// TIA Portal V17 export
// export: Created 2024-08-07T21:44:00.3831212Z, ExportSetting WithDefaults, DisplayName Totally Integrated Automation Portal, DisplayVersion V17 Update 7, DisplayName TIA Portal Openness, DisplayVersion V17 Update 7, DisplayName TIA Portal Version Control Interface, DisplayVersion V17, DisplayName SINAMICS Startdrive Advanced, DisplayVersion V17 SP2, DisplayName SINAMICS Startdrive G110M, G120, G120C, G120D, G120P, G115D, DisplayVersion V17 SP2, DisplayName SINAMICS Startdrive G130, G150, S120, S150, SINAMICS MV, S210, DisplayVersion V17 SP2, DisplayName STEP 7 Professional, DisplayVersion V17 Update 7, DisplayName STEP 7 Safety, DisplayVersion V17 Update 6, DisplayName WinCC Advanced / Unified PC, DisplayVersion V17 Update 7
DATA_BLOCK "DB_EksList"   // DB5051
{ S7_Optimized_Access := 'TRUE' }
VERSION : 0.1
// stored: AutoNumber false, DBAccessibleFromOPCUA true, DBAccessibleFromWebserver true, IsOnlyStoredInLoadMemory false, IsRetainMemResEnabled false, IsWriteProtectedInAS false, MemoryReserve 100
   VAR RETAIN
      Key { S7_SetPoint := 'True'} : Array[1.."EksNumberOfKeys"] of "UDT_EksKey";
   END_VAR
BEGIN
   Key[1..5].Level := 5;
   Key[6..9].Level := 3;
   Key[10..13].Level := 2;
   Key[14..18].Level := 5;
   Key[19..100].Level := 0;
   Key[1].EmployeeID[1..4] := ' ';
   Key[2].EmployeeID[1] := '¥';
   Key[2].EmployeeID[2] := 'Z';
   Key[2].EmployeeID[3] := '¥';
   Key[2].EmployeeID[4] := 'Z';
   Key[3].EmployeeID[1..4] := ' ';
   Key[4].EmployeeID[1..4] := ' ';
   Key[5].EmployeeID[1..4] := ' ';
   Key[6].EmployeeID[1..4] := ' ';
   Key[7].EmployeeID[1..4] := ' ';
   Key[8].EmployeeID[1..4] := ' ';
   Key[9].EmployeeID[1..4] := ' ';
   Key[10].EmployeeID[1..4] := ' ';
   Key[11].EmployeeID[1..4] := ' ';
   Key[12].EmployeeID[1..4] := ' ';
   Key[13].EmployeeID[1..4] := ' ';
   Key[14].EmployeeID[1..4] := ' ';
   Key[15].EmployeeID[1..4] := ' ';
   Key[16].EmployeeID[1..4] := ' ';
   Key[17].EmployeeID[1..4] := ' ';
   Key[18].EmployeeID[1..4] := ' ';
   Key[19].EmployeeID[1..4] := ' ';
   Key[20].EmployeeID[1..4] := ' ';
   Key[21].EmployeeID[1..4] := ' ';
   Key[22].EmployeeID[1..4] := ' ';
   Key[23].EmployeeID[1..4] := ' ';
   Key[24].EmployeeID[1..4] := ' ';
   Key[25].EmployeeID[1..4] := ' ';
   Key[26].EmployeeID[1..4] := ' ';
   Key[27].EmployeeID[1..4] := ' ';
   Key[28].EmployeeID[1..4] := ' ';
   Key[29].EmployeeID[1..4] := ' ';
   Key[30].EmployeeID[1..4] := ' ';
   Key[31].EmployeeID[1..4] := ' ';
   Key[32].EmployeeID[1..4] := ' ';
   Key[33].EmployeeID[1..4] := ' ';
   Key[34].EmployeeID[1..4] := ' ';
   Key[35].EmployeeID[1..4] := ' ';
   Key[36].EmployeeID[1..4] := ' ';
   Key[37].EmployeeID[1..4] := ' ';
   Key[38].EmployeeID[1..4] := ' ';
   Key[39].EmployeeID[1..4] := ' ';
   Key[40].EmployeeID[1..4] := ' ';
   Key[41].EmployeeID[1..4] := ' ';
   Key[42].EmployeeID[1..4] := ' ';
   Key[43].EmployeeID[1..4] := ' ';
   Key[44].EmployeeID[1..4] := ' ';
   Key[45].EmployeeID[1..4] := ' ';
   Key[46].EmployeeID[1..4] := ' ';
   Key[47].EmployeeID[1..4] := ' ';
   Key[48].EmployeeID[1..4] := ' ';
   Key[49].EmployeeID[1..4] := ' ';
   Key[50].EmployeeID[1..4] := ' ';
   Key[51].EmployeeID[1..4] := ' ';
   Key[52].EmployeeID[1..4] := ' ';
   Key[53].EmployeeID[1..4] := ' ';
   Key[54].EmployeeID[1..4] := ' ';
   Key[55].EmployeeID[1..4] := ' ';
   Key[56].EmployeeID[1..4] := ' ';
   Key[57].EmployeeID[1..4] := ' ';
   Key[58].EmployeeID[1..4] := ' ';
   Key[59].EmployeeID[1..4] := ' ';
   Key[60].EmployeeID[1..4] := ' ';
   Key[61].EmployeeID[1..4] := ' ';
   Key[62].EmployeeID[1..4] := ' ';
   Key[63].EmployeeID[1..4] := ' ';
   Key[64].EmployeeID[1..4] := ' ';
   Key[65].EmployeeID[1..4] := ' ';
   Key[66].EmployeeID[1..4] := ' ';
   Key[67].EmployeeID[1..4] := ' ';
   Key[68].EmployeeID[1..4] := ' ';
   Key[69].EmployeeID[1..4] := ' ';
   Key[70].EmployeeID[1..4] := ' ';
   Key[71].EmployeeID[1..4] := ' ';
   Key[72].EmployeeID[1..4] := ' ';
   Key[73].EmployeeID[1..4] := ' ';
   Key[74].EmployeeID[1..4] := ' ';
   Key[75].EmployeeID[1..4] := ' ';
   Key[76].EmployeeID[1..4] := ' ';
   Key[77].EmployeeID[1..4] := ' ';
   Key[78].EmployeeID[1..4] := ' ';
   Key[79].EmployeeID[1..4] := ' ';
   Key[80].EmployeeID[1..4] := ' ';
   Key[81].EmployeeID[1..4] := ' ';
   Key[82].EmployeeID[1..4] := ' ';
   Key[83].EmployeeID[1..4] := ' ';
   Key[84].EmployeeID[1..4] := ' ';
   Key[85].EmployeeID[1..4] := ' ';
   Key[86].EmployeeID[1..4] := ' ';
   Key[87].EmployeeID[1..4] := ' ';
   Key[88].EmployeeID[1..4] := ' ';
   Key[89].EmployeeID[1..4] := ' ';
   Key[90].EmployeeID[1..4] := ' ';
   Key[91].EmployeeID[1..4] := ' ';
   Key[92].EmployeeID[1..4] := ' ';
   Key[93].EmployeeID[1..4] := ' ';
   Key[94].EmployeeID[1..4] := ' ';
   Key[95].EmployeeID[1..4] := ' ';
   Key[96].EmployeeID[1..4] := ' ';
   Key[97].EmployeeID[1..4] := ' ';
   Key[98].EmployeeID[1..4] := ' ';
   Key[99].EmployeeID[1..4] := ' ';
   Key[100].EmployeeID[1..4] := ' ';
   Key[1].KeyID[1] := '0';
   Key[1].KeyID[2] := '3';
   Key[1].KeyID[3] := '6';
   Key[1].KeyID[4] := 'C';
   Key[1].KeyID[5] := 'B';
   Key[1].KeyID[6] := 'C';
   Key[1].KeyID[7] := 'F';
   Key[1].KeyID[8] := '4';
   Key[1].KeyID[9] := '0';
   Key[1].KeyID[10] := 'F';
   Key[1].KeyID[11..12] := '0';
   Key[1].KeyID[13] := '1';
   Key[1].KeyID[14] := '0';
   Key[1].KeyID[15] := '3';
   Key[1].KeyID[16] := '2';
   Key[2].KeyID[1] := '0';
   Key[2].KeyID[2..3] := '3';
   Key[2].KeyID[4] := 'E';
   Key[2].KeyID[5] := '0';
   Key[2].KeyID[6] := '2';
   Key[2].KeyID[7] := 'E';
   Key[2].KeyID[8] := '5';
   Key[2].KeyID[9] := 'C';
   Key[2].KeyID[10] := 'B';
   Key[2].KeyID[11..12] := '0';
   Key[2].KeyID[13] := '1';
   Key[2].KeyID[14] := '0';
   Key[2].KeyID[15] := '3';
   Key[2].KeyID[16] := '2';
   Key[3].KeyID[1] := '0';
   Key[3].KeyID[2] := '3';
   Key[3].KeyID[3] := '7';
   Key[3].KeyID[4] := '2';
   Key[3].KeyID[5] := '4';
   Key[3].KeyID[6] := '5';
   Key[3].KeyID[7] := '2';
   Key[3].KeyID[8] := '9';
   Key[3].KeyID[9] := 'A';
   Key[3].KeyID[10] := '6';
   Key[3].KeyID[11..12] := '0';
   Key[3].KeyID[13] := '1';
   Key[3].KeyID[14] := '0';
   Key[3].KeyID[15] := '3';
   Key[3].KeyID[16] := '2';
   Key[4].KeyID[1] := '0';
   Key[4].KeyID[2] := '3';
   Key[4].KeyID[3] := '7';
   Key[4].KeyID[4] := '2';
   Key[4].KeyID[5..6] := '5';
   Key[4].KeyID[7] := '9';
   Key[4].KeyID[8] := 'D';
   Key[4].KeyID[9] := '8';
   Key[4].KeyID[10] := 'A';
   Key[4].KeyID[11..12] := '0';
   Key[4].KeyID[13] := '1';
   Key[4].KeyID[14] := '0';
   Key[4].KeyID[15] := '3';
   Key[4].KeyID[16] := '2';
   Key[5].KeyID[1] := '0';
   Key[5].KeyID[2] := '3';
   Key[5].KeyID[3] := '7';
   Key[5].KeyID[4] := '2';
   Key[5].KeyID[5] := '4';
   Key[5].KeyID[6] := '3';
   Key[5].KeyID[7] := 'B';
   Key[5].KeyID[8] := 'A';
   Key[5].KeyID[9] := '3';
   Key[5].KeyID[10] := 'F';
   Key[5].KeyID[11..12] := '0';
   Key[5].KeyID[13] := '1';
   Key[5].KeyID[14] := '0';
   Key[5].KeyID[15] := '3';
   Key[5].KeyID[16] := '2';
   Key[6].KeyID[1] := '0';
   Key[6].KeyID[2] := '3';
   Key[6].KeyID[3] := '7';
   Key[6].KeyID[4] := '2';
   Key[6].KeyID[5] := '9';
   Key[6].KeyID[6] := '7';
   Key[6].KeyID[7] := '0';
   Key[6].KeyID[8] := 'C';
   Key[6].KeyID[9] := '2';
   Key[6].KeyID[10] := 'A';
   Key[6].KeyID[11..12] := '0';
   Key[6].KeyID[13] := '1';
   Key[6].KeyID[14] := '0';
   Key[6].KeyID[15] := '3';
   Key[6].KeyID[16] := '2';
   Key[7].KeyID[1] := '0';
   Key[7].KeyID[2] := '3';
   Key[7].KeyID[3] := '7';
   Key[7].KeyID[4] := '3';
   Key[7].KeyID[5] := '0';
   Key[7].KeyID[6] := 'A';
   Key[7].KeyID[7] := 'D';
   Key[7].KeyID[8] := '7';
   Key[7].KeyID[9] := '0';
   Key[7].KeyID[10] := '1';
   Key[7].KeyID[11..12] := '0';
   Key[7].KeyID[13] := '1';
   Key[7].KeyID[14] := '0';
   Key[7].KeyID[15] := '3';
   Key[7].KeyID[16] := '2';
   Key[8].KeyID[1] := '0';
   Key[8].KeyID[2] := '3';
   Key[8].KeyID[3] := '7';
   Key[8].KeyID[4] := '2';
   Key[8].KeyID[5] := '4';
   Key[8].KeyID[6..7] := '5';
   Key[8].KeyID[8..9] := 'F';
   Key[8].KeyID[10] := 'B';
   Key[8].KeyID[11..12] := '0';
   Key[8].KeyID[13] := '1';
   Key[8].KeyID[14] := '0';
   Key[8].KeyID[15] := '3';
   Key[8].KeyID[16] := '2';
   Key[9].KeyID[1] := '0';
   Key[9].KeyID[2] := '3';
   Key[9].KeyID[3] := '7';
   Key[9].KeyID[4] := '2';
   Key[9].KeyID[5] := '9';
   Key[9].KeyID[6] := 'C';
   Key[9].KeyID[7] := '3';
   Key[9].KeyID[8] := '8';
   Key[9].KeyID[9] := '3';
   Key[9].KeyID[10] := '2';
   Key[9].KeyID[11..12] := '0';
   Key[9].KeyID[13] := '1';
   Key[9].KeyID[14] := '0';
   Key[9].KeyID[15] := '3';
   Key[9].KeyID[16] := '2';
   Key[10].KeyID[1] := '0';
   Key[10].KeyID[2] := '3';
   Key[10].KeyID[3] := '7';
   Key[10].KeyID[4] := '2';
   Key[10].KeyID[5] := 'C';
   Key[10].KeyID[6..7] := '3';
   Key[10].KeyID[8] := 'E';
   Key[10].KeyID[9] := 'B';
   Key[10].KeyID[10] := '6';
   Key[10].KeyID[11..12] := '0';
   Key[10].KeyID[13] := '1';
   Key[10].KeyID[14] := '0';
   Key[10].KeyID[15] := '3';
   Key[10].KeyID[16] := '2';
   Key[11].KeyID[1] := '0';
   Key[11].KeyID[2] := '3';
   Key[11].KeyID[3] := '7';
   Key[11].KeyID[4] := '3';
   Key[11].KeyID[5] := '0';
   Key[11].KeyID[6] := 'C';
   Key[11].KeyID[7] := '3';
   Key[11].KeyID[8] := '0';
   Key[11].KeyID[9] := 'B';
   Key[11].KeyID[10] := 'F';
   Key[11].KeyID[11..12] := '0';
   Key[11].KeyID[13] := '1';
   Key[11].KeyID[14] := '0';
   Key[11].KeyID[15] := '3';
   Key[11].KeyID[16] := '2';
   Key[12].KeyID[1] := '0';
   Key[12].KeyID[2] := '3';
   Key[12].KeyID[3] := '7';
   Key[12].KeyID[4] := '2';
   Key[12].KeyID[5] := 'F';
   Key[12].KeyID[6] := '4';
   Key[12].KeyID[7] := 'D';
   Key[12].KeyID[8] := 'F';
   Key[12].KeyID[9] := '5';
   Key[12].KeyID[10] := 'C';
   Key[12].KeyID[11..12] := '0';
   Key[12].KeyID[13] := '1';
   Key[12].KeyID[14] := '0';
   Key[12].KeyID[15] := '3';
   Key[12].KeyID[16] := '2';
   Key[13].KeyID[1] := '0';
   Key[13].KeyID[2] := '3';
   Key[13].KeyID[3] := '7';
   Key[13].KeyID[4] := '2';
   Key[13].KeyID[5] := 'C';
   Key[13].KeyID[6] := '9';
   Key[13].KeyID[7] := '1';
   Key[13].KeyID[8..9] := '6';
   Key[13].KeyID[10] := '7';
   Key[13].KeyID[11..12] := '0';
   Key[13].KeyID[13] := '1';
   Key[13].KeyID[14] := '0';
   Key[13].KeyID[15] := '3';
   Key[13].KeyID[16] := '2';
   Key[14].KeyID[1] := '0';
   Key[14].KeyID[2] := '3';
   Key[14].KeyID[3] := '2';
   Key[14].KeyID[4] := '3';
   Key[14].KeyID[5] := 'C';
   Key[14].KeyID[6] := 'F';
   Key[14].KeyID[7] := '5';
   Key[14].KeyID[8] := 'E';
   Key[14].KeyID[9..10] := 'B';
   Key[14].KeyID[11..12] := '0';
   Key[14].KeyID[13] := '1';
   Key[14].KeyID[14] := '0';
   Key[14].KeyID[15] := '3';
   Key[14].KeyID[16] := '2';
   Key[15].KeyID[1] := '0';
   Key[15].KeyID[2] := '3';
   Key[15].KeyID[3] := '6';
   Key[15].KeyID[4] := '1';
   Key[15].KeyID[5] := 'E';
   Key[15].KeyID[6] := '8';
   Key[15].KeyID[7] := '1';
   Key[15].KeyID[8] := '4';
   Key[15].KeyID[9] := 'A';
   Key[15].KeyID[10] := 'E';
   Key[15].KeyID[11..12] := '0';
   Key[15].KeyID[13] := '1';
   Key[15].KeyID[14] := '0';
   Key[15].KeyID[15] := '3';
   Key[15].KeyID[16] := '2';
   Key[16].KeyID[1] := '0';
   Key[16].KeyID[2] := '3';
   Key[16].KeyID[3] := '7';
   Key[16].KeyID[4] := '1';
   Key[16].KeyID[5] := 'E';
   Key[16].KeyID[6] := 'D';
   Key[16].KeyID[7] := '1';
   Key[16].KeyID[8] := '2';
   Key[16].KeyID[9] := 'B';
   Key[16].KeyID[10] := '7';
   Key[16].KeyID[11..12] := '0';
   Key[16].KeyID[13] := '1';
   Key[16].KeyID[14] := '0';
   Key[16].KeyID[15] := '3';
   Key[16].KeyID[16] := '2';
   Key[17].KeyID[1] := '0';
   Key[17].KeyID[2] := '3';
   Key[17].KeyID[3] := '7';
   Key[17].KeyID[4] := '2';
   Key[17].KeyID[5] := 'F';
   Key[17].KeyID[6] := '5';
   Key[17].KeyID[7] := '2';
   Key[17].KeyID[8] := 'C';
   Key[17].KeyID[9] := '6';
   Key[17].KeyID[10] := '8';
   Key[17].KeyID[11..12] := '0';
   Key[17].KeyID[13] := '1';
   Key[17].KeyID[14] := '0';
   Key[17].KeyID[15] := '3';
   Key[17].KeyID[16] := '2';
   Key[18].KeyID[1] := '0';
   Key[18].KeyID[2] := '3';
   Key[18].KeyID[3] := '7';
   Key[18].KeyID[4] := '1';
   Key[18].KeyID[5..7] := 'F';
   Key[18].KeyID[8] := 'C';
   Key[18].KeyID[9] := '4';
   Key[18].KeyID[10] := '2';
   Key[18].KeyID[11..12] := '0';
   Key[18].KeyID[13] := '1';
   Key[18].KeyID[14] := '0';
   Key[18].KeyID[15] := '3';
   Key[18].KeyID[16] := '2';
   Key[19].KeyID[1..16] := ' ';
   Key[20].KeyID[1..16] := ' ';
   Key[21].KeyID[1..16] := ' ';
   Key[22].KeyID[1..16] := ' ';
   Key[23].KeyID[1..16] := ' ';
   Key[24].KeyID[1..16] := ' ';
   Key[25].KeyID[1..16] := ' ';
   Key[26].KeyID[1..16] := ' ';
   Key[27].KeyID[1..16] := ' ';
   Key[28].KeyID[1..16] := ' ';
   Key[29].KeyID[1..16] := ' ';
   Key[30].KeyID[1..16] := ' ';
   Key[31].KeyID[1..16] := ' ';
   Key[32].KeyID[1..16] := ' ';
   Key[33].KeyID[1..16] := ' ';
   Key[34].KeyID[1..16] := ' ';
   Key[35].KeyID[1..16] := ' ';
   Key[36].KeyID[1..16] := ' ';
   Key[37].KeyID[1..16] := ' ';
   Key[38].KeyID[1..16] := ' ';
   Key[39].KeyID[1..16] := ' ';
   Key[40].KeyID[1..16] := ' ';
   Key[41].KeyID[1..16] := ' ';
   Key[42].KeyID[1..16] := ' ';
   Key[43].KeyID[1..16] := ' ';
   Key[44].KeyID[1..16] := ' ';
   Key[45].KeyID[1..16] := ' ';
   Key[46].KeyID[1..16] := ' ';
   Key[47].KeyID[1..16] := ' ';
   Key[48].KeyID[1..16] := ' ';
   Key[49].KeyID[1..16] := ' ';
   Key[50].KeyID[1..16] := ' ';
   Key[51].KeyID[1..16] := ' ';
   Key[52].KeyID[1..16] := ' ';
   Key[53].KeyID[1..16] := ' ';
   Key[54].KeyID[1..16] := ' ';
   Key[55].KeyID[1..16] := ' ';
   Key[56].KeyID[1..16] := ' ';
   Key[57].KeyID[1..16] := ' ';
   Key[58].KeyID[1..16] := ' ';
   Key[59].KeyID[1..16] := ' ';
   Key[60].KeyID[1..16] := ' ';
   Key[61].KeyID[1..16] := ' ';
   Key[62].KeyID[1..16] := ' ';
   Key[63].KeyID[1..16] := ' ';
   Key[64].KeyID[1..16] := ' ';
   Key[65].KeyID[1..16] := ' ';
   Key[66].KeyID[1..16] := ' ';
   Key[67].KeyID[1..16] := ' ';
   Key[68].KeyID[1..16] := ' ';
   Key[69].KeyID[1..16] := ' ';
   Key[70].KeyID[1..16] := ' ';
   Key[71].KeyID[1..16] := ' ';
   Key[72].KeyID[1..16] := ' ';
   Key[73].KeyID[1..16] := ' ';
   Key[74].KeyID[1..16] := ' ';
   Key[75].KeyID[1..16] := ' ';
   Key[76].KeyID[1..16] := ' ';
   Key[77].KeyID[1..16] := ' ';
   Key[78].KeyID[1..16] := ' ';
   Key[79].KeyID[1..16] := ' ';
   Key[80].KeyID[1..16] := ' ';
   Key[81].KeyID[1..16] := ' ';
   Key[82].KeyID[1..16] := ' ';
   Key[83].KeyID[1..16] := ' ';
   Key[84].KeyID[1..16] := ' ';
   Key[85].KeyID[1..16] := ' ';
   Key[86].KeyID[1..16] := ' ';
   Key[87].KeyID[1..16] := ' ';
   Key[88].KeyID[1..16] := ' ';
   Key[89].KeyID[1..16] := ' ';
   Key[90].KeyID[1..16] := ' ';
   Key[91].KeyID[1..16] := ' ';
   Key[92].KeyID[1..16] := ' ';
   Key[93].KeyID[1..16] := ' ';
   Key[94].KeyID[1..16] := ' ';
   Key[95].KeyID[1..16] := ' ';
   Key[96].KeyID[1..16] := ' ';
   Key[97].KeyID[1..16] := ' ';
   Key[98].KeyID[1..16] := ' ';
   Key[99].KeyID[1..16] := ' ';
   Key[100].KeyID[1..16] := ' ';
   Key[1].Comment[1..20] := ' ';
   Key[2].Comment[1..20] := ' ';
   Key[3].Comment[1..20] := ' ';
   Key[4].Comment[1..20] := ' ';
   Key[5].Comment[1..20] := ' ';
   Key[6].Comment[1..20] := ' ';
   Key[7].Comment[1..20] := ' ';
   Key[8].Comment[1..20] := ' ';
   Key[9].Comment[1..20] := ' ';
   Key[10].Comment[1..20] := ' ';
   Key[11].Comment[1..20] := ' ';
   Key[12].Comment[1..20] := ' ';
   Key[13].Comment[1..20] := ' ';
   Key[14].Comment[1..20] := ' ';
   Key[15].Comment[1..20] := ' ';
   Key[16].Comment[1..20] := ' ';
   Key[17].Comment[1..20] := ' ';
   Key[18].Comment[1..20] := ' ';
   Key[19].Comment[1..20] := ' ';
   Key[20].Comment[1..20] := ' ';
   Key[21].Comment[1..20] := ' ';
   Key[22].Comment[1..20] := ' ';
   Key[23].Comment[1..20] := ' ';
   Key[24].Comment[1..20] := ' ';
   Key[25].Comment[1..20] := ' ';
   Key[26].Comment[1..20] := ' ';
   Key[27].Comment[1..20] := ' ';
   Key[28].Comment[1..20] := ' ';
   Key[29].Comment[1..20] := ' ';
   Key[30].Comment[1..20] := ' ';
   Key[31].Comment[1..20] := ' ';
   Key[32].Comment[1..20] := ' ';
   Key[33].Comment[1..20] := ' ';
   Key[34].Comment[1..20] := ' ';
   Key[35].Comment[1..20] := ' ';
   Key[36].Comment[1..20] := ' ';
   Key[37].Comment[1..20] := ' ';
   Key[38].Comment[1..20] := ' ';
   Key[39].Comment[1..20] := ' ';
   Key[40].Comment[1..20] := ' ';
   Key[41].Comment[1..20] := ' ';
   Key[42].Comment[1..20] := ' ';
   Key[43].Comment[1..20] := ' ';
   Key[44].Comment[1..20] := ' ';
   Key[45].Comment[1..20] := ' ';
   Key[46].Comment[1..20] := ' ';
   Key[47].Comment[1..20] := ' ';
   Key[48].Comment[1..20] := ' ';
   Key[49].Comment[1..20] := ' ';
   Key[50].Comment[1..20] := ' ';
   Key[51].Comment[1..20] := ' ';
   Key[52].Comment[1..20] := ' ';
   Key[53].Comment[1..20] := ' ';
   Key[54].Comment[1..20] := ' ';
   Key[55].Comment[1..20] := ' ';
   Key[56].Comment[1..20] := ' ';
   Key[57].Comment[1..20] := ' ';
   Key[58].Comment[1..20] := ' ';
   Key[59].Comment[1..20] := ' ';
   Key[60].Comment[1..20] := ' ';
   Key[61].Comment[1..20] := ' ';
   Key[62].Comment[1..20] := ' ';
   Key[63].Comment[1..20] := ' ';
   Key[64].Comment[1..20] := ' ';
   Key[65].Comment[1..20] := ' ';
   Key[66].Comment[1..20] := ' ';
   Key[67].Comment[1..20] := ' ';
   Key[68].Comment[1..20] := ' ';
   Key[69].Comment[1..20] := ' ';
   Key[70].Comment[1..20] := ' ';
   Key[71].Comment[1..20] := ' ';
   Key[72].Comment[1..20] := ' ';
   Key[73].Comment[1..20] := ' ';
   Key[74].Comment[1..20] := ' ';
   Key[75].Comment[1..20] := ' ';
   Key[76].Comment[1..20] := ' ';
   Key[77].Comment[1..20] := ' ';
   Key[78].Comment[1..20] := ' ';
   Key[79].Comment[1..20] := ' ';
   Key[80].Comment[1..20] := ' ';
   Key[81].Comment[1..20] := ' ';
   Key[82].Comment[1..20] := ' ';
   Key[83].Comment[1..20] := ' ';
   Key[84].Comment[1..20] := ' ';
   Key[85].Comment[1..20] := ' ';
   Key[86].Comment[1..20] := ' ';
   Key[87].Comment[1..20] := ' ';
   Key[88].Comment[1..20] := ' ';
   Key[89].Comment[1..20] := ' ';
   Key[90].Comment[1..20] := ' ';
   Key[91].Comment[1..20] := ' ';
   Key[92].Comment[1..20] := ' ';
   Key[93].Comment[1..20] := ' ';
   Key[94].Comment[1..20] := ' ';
   Key[95].Comment[1..20] := ' ';
   Key[96].Comment[1..20] := ' ';
   Key[97].Comment[1..20] := ' ';
   Key[98].Comment[1..20] := ' ';
   Key[99].Comment[1..20] := ' ';
   Key[100].Comment[1..20] := ' ';
END_DATA_BLOCK
